(* Schneider Machine Expert - Basic project Nuevo proyecto, file version 2.8.0.0 *)
(* ProjectInformations: Name=Nuevo proyecto *)

HARDWARE
  Cpu 0: TM221CE24T
  EthernetConfiguration: NetworkName=M221, IpAllocationMode=FixedAddress, IpAddress=192.168.13.63, SubnetMask=255.255.255.0
  SerialLineConfiguration: Baud=Baud19200, Parity=ParityNone, DataBits=DataBits8, StopBits=StopBits1, PhysicalMedium=PhysicalMediumRs485, TransmissionMode=TransmissionModeModbusRtu, SlaveId=1, Addressing=MasterAddressing
  MastTask: UsePeriodScanMode=false, PeriodScan=100
  FastTask: Period=255
  CpuBehavior: StartingMode=StartAsPreviousState, AutoSaveRamOnEeprom=true, WatchdogPeriod=500

SYMBOLS  (address, symbol, comment, settings)
  %S6       SB_TB1S  "Base de tiempo de 1 s generada por un reloj interno"
  %READ_VAR0   [Link(Value(FBComLinkParameterEnums=SerialLine1)), RemoteDeviceId(Value(int=1)), Timeout(Value(int=250)), ObjType(Value(FBComObjTypeParameterEnums=MW)), FirstObj(Value(int=8959)), Quantity(Value(int=4)), IndexData(Value(int=0))]
  %WRITE_VAR0   [Link(Value(FBComLinkParameterEnums=SerialLine1)), RemoteDeviceId(Value(int=1)), Timeout(Value(int=250)), ObjType(Value(FBComObjTypeParameterEnums=MW)), FirstObj(Value(int=8959)), Quantity(Value(int=4)), IndexData(Value(int=0))]

POU Nuevo POU
  (* SectionNumber=1 *)

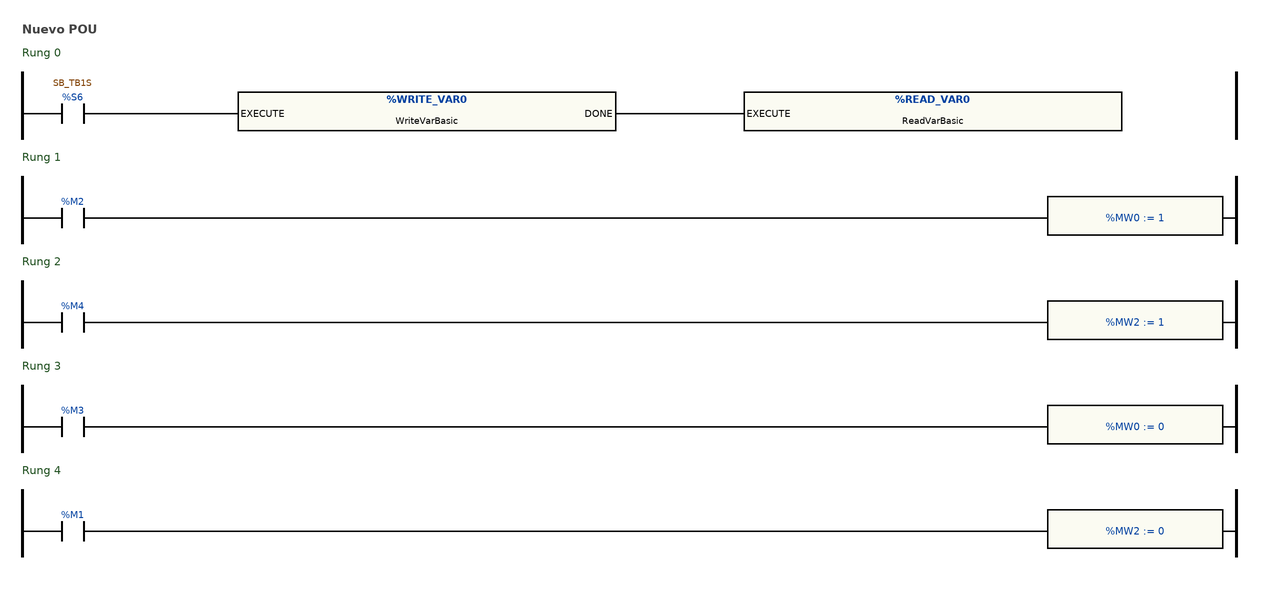

// Rung 0
  LD 1
  MULTIFB
  BLK %WRITE_VAR0
  LD %S6                  (* SB_TB1S *)
  EXECUTE
  OUT_BLK
  LD DONE
  ST %MW2009:X0
  END_BLK
  BLK %READ_VAR0
  LD %MW2009:X0
  EXECUTE
  END_BLK
  MULTIFB
  // as ST:
  //   %WRITE_VAR0(EXECUTE := SB_TB1S);
  //   %READ_VAR0(EXECUTE := %WRITE_VAR0.DONE);

// Rung 1
  LD %M2
  [ %MW0 := 1 ]
  // as ST:
  //   IF %M2 THEN %MW0 := 1; END_IF;

// Rung 2
  LD %M4
  [ %MW2 := 1 ]
  // as ST:
  //   IF %M4 THEN %MW2 := 1; END_IF;

// Rung 3
  LD %M3
  [ %MW0 := 0 ]
  // as ST:
  //   IF %M3 THEN %MW0 := 0; END_IF;

// Rung 4
  LD %M1
  [ %MW2 := 0 ]
  // as ST:
  //   IF %M1 THEN %MW2 := 0; END_IF;
